/// Move the TCP relative to a reference cartesian position (PTPT interpolation)
FUNCTION_BLOCK MoveDirectOffsetFB EXTENDS RobotLibraryBaseFB
// ------------------------------------------------------------------------- 
//  SRCI Robot Library                                                
// ------------------------------------------------------------------------- 
//                                                                           
//  Object:      MoveDirectOffsetFB                                       
//  Author:      Thorsten Brach                                                
//  Date:        2024-06-01
//
//  Description:                                              
//   
//                                                                           
//  Copyright: 
//    (C) 2024 Thorsten Brach. All rights reserved                                                                         
//                                                                           
//  Disclaimer:                                                                           
//    This project is provided without any guarantee and can be used for   
//    private and commercial purposes. Any commercial use is at the user’s 
//    own risk and responsibility.
//
// -------------------------------------------------------------------------
VAR_INPUT
  /// Start of the command at the rising edge
  Execute            : BOOL;
  /// Absolute reference coordinates in the selected coordinate system (see input parameters ToolNo and FrameNo).
  ReferencePosition  : RobotCartesianPosition;
  /// Relative distance and rotation from ReferencePosition.
  Offset             : RobotCartesianPosition;
  /// Defines type of reference coordinate system of the offset position
  ReferenceType      : ReferenceType;
  /// TCP velocity in % of nominal velocity
  /// •  <0%: (default) - Use default velocity
  /// •   0%:           - Use internal minimal velocity
  /// • 100%:           - Use maximal reference velocity
  /// See chapter 5.5.7 Robot dynamics
  VelocityRate       : REAL;
  /// Acceleration for movement in % of nominal acceleration
  /// •  <0%: (default) - Use default acceleration
  /// •   0%:           - Use internal minimal acceleration
  /// • 100%:           - Use maximal reference acceleration
  /// See chapter 5.5.7 Robot dynamics
  AccelerationRate   : REAL;
  /// Deceleration for movement in % of nominal deceleration
  /// •  <0%: (default) - Use default deceleration 
  /// •   0%:           - Use internal minimal deceleration
  /// • 100%:           - Use maximal reference deceleration
  /// See chapter 5.5.7 Robot dynamics
  DecelerationRate   : REAL;
  /// Jerk of the movement in % of nominal jerk
  /// •  <0%: (default) - Use default jerk
  /// •   0%:           - Use internal minimal jerk
  /// • 100%:           - Use maximal reference jerk
  /// See chapter 5.5.7 Robot dynamics
  JerkRate           : REAL;
  /// Index of tool
  /// •      0: Flange (default)
  /// • 1..254: Tool frames
  ToolNo             : USINT;
  /// Index of frame
  /// •      0: WCS (default)
  /// • 1..254: User frames
  FrameNo            : USINT;
  /// Parameter which determines the behavior towards the previously sent and still active or buffered commands
  AbortingMode       : AbortingMode;
  /// Parameter which determines the transition behavior at the end of the movement to be sent to the next command. 
  /// The user can choose a transition type between exact stop and different blend possibilities
  BlendingMode       : BlendingMode;
  /// Additional parameter for the blending mode, to define i.e. velocity limit (%) or blending radius
  BlendingParameter  : ARRAY [0..1] OF REAL := [10,0];
  /// Parameter is used if it is greater than 0 (default)
  /// • Velocity input is ignored
  /// • Parameter defines the time for the movement to reach the target position
  /// Error is sent by the RC if the time cannot be kept
  MoveTime           : TIME;
  /// Parameter to describe how the orientation axes (RX, RY, RZ) will be interpolated during the movement.
  OriMode            : OriMode;
  /// Defines the usage of the config byte inside the position according to Table 6-238
  ConfigMode         : ArmConfigParameter;
  /// Defines the usage of the TurnNumber byte inside the position.
  TurnMode           : TurnMode;
  /// Set TRUE to allow manipulation of this move command through superimposing functions.
  /// For more information see chapter 5.5.9.5
  Manipulation       : BOOL;
  /// Defines the target sequence in which the command will be executed
  SequenceFlag       : SequenceFlag;
  /// ID of Action that will be executed when this command is active
  /// • >0: Start Action - Start executing the Action function with the identical ListenerID.
  /// • <0: Stop Action  -  Stop executing the Action function with the identical ListenerID.
  /// • 0: No trigger (default)-  If no EmitterID is defined, the function will not trigger any Action during its execution
  /// For more information see section Triggers of this chapter or chapter 5.5.12.4.
  EmitterID          : ARRAY [0..3] OF SINT;
END_VAR

VAR_OUTPUT
  /// The command has been completed successfully
  Done               : BOOL;
  /// FB is being processed
  Busy               : BOOL;
  /// Command is transferred and confirmed by the RC
  CommandBuffered    : BOOL;
  /// The command takes control of the motion of the according axis group
  Active             : BOOL;
  /// The command was aborted by another command.
  CommandAborted     : BOOL;
  /// TRUE, while command is interrupted during execution and can be continued
  CommandInterrupted : BOOL;
  /// Distance-to-go of the current job.
  /// • -1: No valid value because move command is not yet active (valid values are pending) or not supported by RC
  /// • >0: Actual distance between current and target position
  /// •  0: Target position reached
  RemainingDistance  : REAL;
  /// Percentage of already traversed distance of current job.
  /// If not supported : • -1
  Progress           : REAL;
  /// Unique system-generated ID of the trigger function when the function is called by the user.
  /// For more information see chapter 5.5.12.4.
  FollowID           : DINT;
END_VAR

                  
                

METHOD PROTECTED OnCall
VAR_IN_OUT
  /// Robot assignment of function
  AxesGroup         : AxesGroup; 
END_VAR
                        
                      
END_METHOD
END_FUNCTION_BLOCK

/// Move Joints relative to relative cartesian position (Relative cartesian PTP) (Joint interpolated movement)
FUNCTION_BLOCK MoveDirectRelativeFB EXTENDS RobotLibraryBaseFB
// ------------------------------------------------------------------------- 
//  SRCI Robot Library                                                
// ------------------------------------------------------------------------- 
//                                                                           
//  Object:      MoveDirectRelativeFB                                       
//  Author:      Thorsten Brach                                                
//  Date:        2024-06-01
//
//  Description:                                              
//   
//                                                                           
//  Copyright: 
//    (C) 2024 Thorsten Brach. All rights reserved                                                                         
//                                                                           
//  Disclaimer:                                                                           
//    This project is provided without any guarantee and can be used for   
//    private and commercial purposes. Any commercial use is at the user’s 
//    own risk and responsibility.
//
// -------------------------------------------------------------------------
VAR_INPUT
  /// Start of the command at the rising edge
  Execute            : BOOL;
  /// Relative distance and rotation from the current or last target position to the end point.
  Distance           : RobotCartesianPosition;
  /// Defines type of reference coordinate system of the offset position 
  ReferenceType      : ReferenceType;
  /// TCP velocity in % of nominal velocity
  /// •  <0%: (default) - Use default velocity
  /// •   0%:           - Use internal minimal velocity
  /// • 100%:           - Use maximal reference velocity
  /// See chapter 5.5.7 Robot dynamics
  ///
  VelocityRate       : REAL;
  /// Acceleration for movement in % of nominal acceleration
  /// •  <0%: (default) - Use default acceleration
  /// •   0%:           - Use internal minimal acceleration
  /// • 100%:           - Use maximal reference acceleration
  /// See chapter 5.5.7 Robot dynamics
  AccelerationRate   : REAL;
  /// Deceleration for movement in % of nominal deceleration
  /// •  <0%: (default) - Use default deceleration 
  /// •   0%:           - Use internal minimal deceleration
  /// • 100%:           - Use maximal reference deceleration
  /// See chapter 5.5.7 Robot dynamics
  DecelerationRate   : REAL;
  /// Jerk of the movement in % of nominal jerk
  /// •  <0%: (default) - Use default jerk
  /// •   0%:           - Use internal minimal jerk
  /// • 100%:           - Use maximal reference jerk
  /// See chapter 5.5.7 Robot dynamics
  JerkRate           : REAL;
  /// Index of tool
  /// •      0: Flange (default)
  /// • 1..254: Tool frames
  ToolNo             : USINT;
  /// Index of frame
  /// •      0: WCS (default)
  /// • 1..254: User frames
  FrameNo            : USINT;
  /// Parameter which determines the behavior towards the previously sent and still active or buffered commands
  AbortingMode       : AbortingMode;
  /// Parameter which determines the transition behavior at the end of the movement to be sent to the next command. 
  /// The user can choose a transition type between exact stop and different blend possibilities
  BlendingMode       : BlendingMode;
  /// Additional parameter for the blending mode, to define i.e. velocity limit (%) or blending radius
  BlendingParameter  : ARRAY [0..1] OF REAL := [10,0];
  /// Parameter is used if it is greater than 0 (default)
  /// • Velocity input is ignored
  /// • Parameter defines the time for the movement to reach the target position
  /// Error is sent by the RC if the time cannot be kept
  MoveTime           : TIME;
  /// Defines the usage of the config byte inside the position according to Table 6-238
  ConfigMode         : ArmConfigParameter;
  /// Defines the usage of the TurnNumber byte inside the position.
  TurnMode           : TurnMode;
  /// Set TRUE to allow manipulation of this move command through superimposing functions.
  /// For more information see chapter 5.5.9.5
  Manipulation       : BOOL;
  /// Defines the target sequence in which the command will be executed
  SequenceFlag       : SequenceFlag;
  /// ID of Action that will be executed when this command is active
  /// • >0: Start Action - Start executing the Action function with the identical ListenerID.
  /// • <0: Stop Action  -  Stop executing the Action function with the identical ListenerID.
  /// • 0: No trigger (default)-  If no EmitterID is defined, the function will not trigger any Action during its execution
  /// For more information see section Triggers of this chapter or chapter 5.5.12.4.
  EmitterID          : ARRAY [0..3] OF SINT;
END_VAR

VAR_OUTPUT
  /// The command has been completed successfully
  Done               : BOOL;
  /// FB is being processed
  Busy               : BOOL;
  /// Command is transferred and confirmed by the RC
  CommandBuffered    : BOOL;
  /// The command takes control of the motion of the according axis group
  Active             : BOOL;
  /// The command was aborted by another command.
  CommandAborted     : BOOL;
  /// TRUE, while command is interrupted during execution and can be continued
  CommandInterrupted : BOOL;
  /// Distance-to-go of the current job.
  /// • -1: No valid value because move command is not yet active (valid values are pending) or not supported by RC
  /// • >0: Actual distance between current and target position
  /// •  0: Target position reached
  RemainingDistance  : REAL;
  /// Percentage of already traversed distance of current job.
  /// If not supported : • -1
  Progress           : REAL;
  /// Unique system-generated ID of the trigger function when the function is called by the user.
  /// For more information see chapter 5.5.12.4.
  FollowID           : DINT;
END_VAR

                  
                

METHOD PROTECTED OnCall
VAR_IN_OUT
  /// Robot assignment of function
  AxesGroup         : AxesGroup; 
END_VAR
                        
                      
END_METHOD
END_FUNCTION_BLOCK

/// Move the TCP to an absolute cartesian position (linear interpolation)
FUNCTION_BLOCK MoveLinearAbsoluteFB EXTENDS RobotLibraryBaseFB
// ------------------------------------------------------------------------- 
//  SRCI Robot Library                                                
// ------------------------------------------------------------------------- 
//                                                                           
//  Object:      MoveLinearAbsoluteFB                                       
//  Author:      Thorsten Brach                                                
//  Date:        2024-06-01
//
//  Description:                                              
//   
//                                                                           
//  Copyright: 
//    (C) 2024 Thorsten Brach. All rights reserved                                                                         
//                                                                           
//  Disclaimer:                                                                           
//    This project is provided without any guarantee and can be used for   
//    private and commercial purposes. Any commercial use is at the user’s 
//    own risk and responsibility.
//
// -------------------------------------------------------------------------
VAR_INPUT
  /// Start of the command at the rising edge
  Execute            : BOOL;
  /// Absolute target coordinates in the selected coordinate system (see input parameters ToolNo and FrameNo)
  Position           : RobotCartesianPosition;
  /// TCP velocity in % of nominal velocity
  /// •  <0%: (default) - Use default velocity
  /// •   0%:           - Use internal minimal velocity
  /// • 100%:           - Use maximal reference velocity
  /// See chapter 5.5.7 Robot dynamics
  VelocityRate       : REAL;
  /// Acceleration for movement in % of nominal acceleration
  /// •  <0%: (default) - Use default acceleration
  /// •   0%:           - Use internal minimal acceleration
  /// • 100%:           - Use maximal reference acceleration
  /// See chapter 5.5.7 Robot dynamics
  AccelerationRate   : REAL;
  /// Deceleration for movement in % of nominal deceleration
  /// •  <0%: (default) - Use default deceleration 
  /// •   0%:           - Use internal minimal deceleration
  /// • 100%:           - Use maximal reference deceleration
  /// See chapter 5.5.7 Robot dynamics
  DecelerationRate   : REAL;
  /// Jerk of the movement in % of nominal jerk
  /// •  <0%: (default) - Use default jerk
  /// •   0%:           - Use internal minimal jerk
  /// • 100%:           - Use maximal reference jerk
  /// See chapter 5.5.7 Robot dynamics
  JerkRate           : REAL;
  /// Index of tool
  /// •      0: Flange (default)
  /// • 1..254: Tool frames
  ToolNo             : USINT;
  /// Index of frame
  /// •      0: WCS (default)
  /// • 1..254: User frames
  FrameNo            : USINT;
  /// Parameter which determines the behavior towards the previously sent and still active or buffered commands
  AbortingMode       : AbortingMode;
  /// Parameter which determines the transition behavior at the end of the movement to be sent to the next command. 
  /// The user can choose a transition type between exact stop and different blend possibilities
  BlendingMode       : BlendingMode;
  /// Additional parameter for the blending mode, to define i.e. velocity limit (%) or blending radius
  BlendingParameter  : ARRAY [0..1] OF REAL := [10,0];
  /// Parameter is used if it is greater than 0 (default)
  /// • Velocity input is ignored
  /// • Parameter defines the time for the movement to reach the target position
  /// Error is sent by the RC if the time cannot be kept
  MoveTime           : TIME;
  /// Parameter to describe how the orientation axes (RX, RY, RZ) will be interpolated during the movement
  OriMode            : OriMode;
  /// Defines the usage of the config byte inside the position according to Table 6-238
  ConfigMode         : ArmConfigParameter;
  /// Defines the usage of the TurnNumber byte inside the position.
  TurnMode           : TurnMode;
  /// Set TRUE to allow manipulation of this move command through superimposing functions.
  /// For more information see chapter 5.5.9.5
  Manipulation       : BOOL;
  /// Defines the target sequence in which the command will be executed
  SequenceFlag       : SequenceFlag;
  /// ID of Action that will be executed when this command is active
  /// • >0: Start Action - Start executing the Action function with the identical ListenerID.
  /// • <0: Stop Action  -  Stop executing the Action function with the identical ListenerID.
  /// • 0: No trigger (default)-  If no EmitterID is defined, the function will not trigger any Action during its execution
  /// For more information see section Triggers of this chapter or chapter 5.5.12.4.
  EmitterID          : ARRAY [0..3] OF SINT;
END_VAR

VAR_OUTPUT
  /// The command has been completed successfully
  Done               : BOOL;
  /// FB is being processed
  Busy               : BOOL;
  /// Command is transferred and confirmed by the RC
  CommandBuffered    : BOOL;
  /// The command takes control of the motion of the according axis group
  Active             : BOOL;
  /// The command was aborted by another command.
  CommandAborted     : BOOL;
  /// TRUE, while command is interrupted during execution and can be continued
  CommandInterrupted : BOOL;
  /// Distance-to-go of the current job.
  /// • -1: No valid value because move command is not yet active (valid values are pending) or not supported by RC
  /// • >0: Actual distance between current and target position
  /// •  0: Target position reached
  RemainingDistance  : REAL;
  /// Percentage of already traversed distance of current job.
  /// If not supported : • -1
  Progress           : REAL;
  /// Unique system-generated ID of the trigger function when the function is called by the user.
  /// For more information see chapter 5.5.12.4.
  FollowID           : DINT;
END_VAR

                  
                

METHOD PROTECTED OnCall
VAR_IN_OUT
  /// Robot assignment of function
  AxesGroup         : AxesGroup; 
END_VAR
                        
                      
END_METHOD
END_FUNCTION_BLOCK

/// Move TCP to an absolute joint position (linear interpolation)
FUNCTION_BLOCK MoveLinearAbsoluteJFB EXTENDS RobotLibraryBaseFB
// ------------------------------------------------------------------------- 
//  SRCI Robot Library                                                
// ------------------------------------------------------------------------- 
//                                                                           
//  Object:      MoveLinearAbsoluteJFB                                       
//  Author:      Thorsten Brach                                                
//  Date:        2024-06-01
//
//  Description:                                              
//   
//                                                                           
//  Copyright: 
//    (C) 2024 Thorsten Brach. All rights reserved                                                                         
//                                                                           
//  Disclaimer:                                                                           
//    This project is provided without any guarantee and can be used for   
//    private and commercial purposes. Any commercial use is at the user’s 
//    own risk and responsibility.
//
// -------------------------------------------------------------------------
VAR_INPUT
  /// Start of the command at the rising edge
  Execute            : BOOL;
  /// Absolute end position of the robot in Joint position.
  JointPosition      : RobotJointPosition;
  /// TCP velocity in % of nominal velocity
  /// •  <0%: (default) - Use default velocity
  /// •   0%:           - Use internal minimal velocity
  /// • 100%:           - Use maximal reference velocity
  /// See chapter 5.5.7 Robot dynamics
  VelocityRate       : REAL;
  /// Acceleration for movement in % of nominal acceleration
  /// •  <0%: (default) - Use default acceleration
  /// •   0%:           - Use internal minimal acceleration
  /// • 100%:           - Use maximal reference acceleration
  /// See chapter 5.5.7 Robot dynamics
  AccelerationRate   : REAL;
  /// Deceleration for movement in % of nominal deceleration
  /// •  <0%: (default) - Use default deceleration 
  /// •   0%:           - Use internal minimal deceleration
  /// • 100%:           - Use maximal reference deceleration
  /// See chapter 5.5.7 Robot dynamics
  DecelerationRate   : REAL;
  /// Jerk of the movement in % of nominal jerk
  /// •  <0%: (default) - Use default jerk
  /// •   0%:           - Use internal minimal jerk
  /// • 100%:           - Use maximal reference jerk
  /// See chapter 5.5.7 Robot dynamics
  JerkRate           : REAL;
  /// Index of tool
  /// •      0: Flange (default)
  /// • 1..254: Tool frames
  ToolNo             : USINT;
  /// Parameter which determines the behavior towards the previously sent and still active or buffered commands
  AbortingMode       : AbortingMode;
  /// Parameter which determines the transition behavior at the end of the movement to be sent to the next command. 
  /// The user can choose a transition type between exact stop and different blend possibilities
  BlendingMode       : BlendingMode;
  /// Additional parameter for the blending mode, to define i.e. velocity limit (%) or blending radius
  BlendingParameter  : ARRAY [0..1] OF REAL := [10,0];
  /// Parameter is used if it is greater than 0 (default)
  /// • Velocity input is ignored
  /// • Parameter defines the time for the movement to reach the target position
  /// Error is sent by the RC if the time cannot be kept
  MoveTime           : TIME;
  /// Parameter to describe how the orientation axes (RX, RY, RZ) will be interpolated during the movement
  OriMode            : OriMode;
  /// Set TRUE to allow manipulation of this move command through superimposing functions.
  /// For more information see chapter 5.5.9.5
  Manipulation       : BOOL;
  /// Defines the target sequence in which the command will be executed
  SequenceFlag       : SequenceFlag;
  /// ID of Action that will be executed when this command is active
  /// • >0: Start Action - Start executing the Action function with the identical ListenerID.
  /// • <0: Stop Action  -  Stop executing the Action function with the identical ListenerID.
  /// • 0: No trigger (default)-  If no EmitterID is defined, the function will not trigger any Action during its execution
  /// For more information see section Triggers of this chapter or chapter 5.5.12.4.
  EmitterID          : ARRAY [0..3] OF SINT;
END_VAR

VAR_OUTPUT
  /// The command has been completed successfully
  Done               : BOOL;
  /// FB is being processed
  Busy               : BOOL;
  /// Command is transferred and confirmed by the RC
  CommandBuffered    : BOOL;
  /// The command takes control of the motion of the according axis group
  Active             : BOOL;
  /// The command was aborted by another command.
  CommandAborted     : BOOL;
  /// TRUE, while command is interrupted during execution and can be continued
  CommandInterrupted : BOOL;
  /// Distance-to-go of the current job.
  /// • -1: No valid value because move command is not yet active (valid values are pending) or not supported by RC
  /// • >0: Actual distance between current and target position
  /// •  0: Target position reached
  RemainingDistance  : REAL;
  /// Percentage of already traversed distance of current job.
  /// If not supported : • -1
  Progress           : REAL;
  /// Unique system-generated ID of the trigger function when the function is called by the user.
  /// For more information see chapter 5.5.12.4.
  FollowID           : DINT;
END_VAR

                  
                

METHOD PROTECTED OnCall
VAR_IN_OUT
  /// Robot assignment of function
  AxesGroup         : AxesGroup; 
END_VAR
                        
                      
END_METHOD
END_FUNCTION_BLOCK

/// Set trigger in defined position of path (L = Linear Path) (cartesian) switch periphery.
FUNCTION_BLOCK MoveLinearCamFB EXTENDS RobotLibraryBaseFB
// ------------------------------------------------------------------------- 
//  SRCI Robot Library                                                
// ------------------------------------------------------------------------- 
//                                                                           
//  Object:      MoveLinearCamFB                                       
//  Author:      Thorsten Brach                                                
//  Date:        2024-06-01
//
//  Description:                                              
//   
//                                                                           
//  Copyright: 
//    (C) 2024 Thorsten Brach. All rights reserved                                                                         
//                                                                           
//  Disclaimer:                                                                           
//    This project is provided without any guarantee and can be used for   
//    private and commercial purposes. Any commercial use is at the user’s 
//    own risk and responsibility.
//
// -------------------------------------------------------------------------
VAR_INPUT
  /// Start of the command at the rising edge
  Execute            : BOOL;
  /// Absolute target coordinates in the selected coordinate system (see input parameters ToolNo and FrameNo)
  Position           : RobotCartesianPosition;
  /// TCP velocity in % of nominal velocity
  /// •  <0%: (default) - Use default velocity
  /// •   0%:           - Use internal minimal velocity
  /// • 100%:           - Use maximal reference velocity
  /// See chapter 5.5.7 Robot dynamics
  VelocityRate       : REAL;
  /// Acceleration for movement in % of nominal acceleration
  /// •  <0%: (default) - Use default acceleration
  /// •   0%:           - Use internal minimal acceleration
  /// • 100%:           - Use maximal reference acceleration
  /// See chapter 5.5.7 Robot dynamics
  AccelerationRate   : REAL;
  /// Deceleration for movement in % of nominal deceleration
  /// •  <0%: (default) - Use default deceleration 
  /// •   0%:           - Use internal minimal deceleration
  /// • 100%:           - Use maximal reference deceleration
  /// See chapter 5.5.7 Robot dynamics
  DecelerationRate   : REAL;
  /// Jerk of the movement in % of nominal jerk
  /// •  <0%: (default) - Use default jerk
  /// •   0%:           - Use internal minimal jerk
  /// • 100%:           - Use maximal reference jerk
  /// See chapter 5.5.7 Robot dynamics
  JerkRate           : REAL;
  /// Index of tool
  /// •      0: Flange (default)
  /// • 1..254: Tool frames
  ToolNo             : USINT;
  /// Index of frame
  /// •      0: WCS (default)
  /// • 1..254: User frames
  FrameNo            : USINT;
  /// Parameter which determines the behavior towards the previously sent and still active or buffered commands
  AbortingMode       : AbortingMode;
  /// Parameter which determines the transition behavior at the end of the movement to be sent to the next command. 
  /// The user can choose a transition type between exact stop and different blend possibilities
  BlendingMode       : BlendingMode;
  /// Additional parameter for the blending mode, to define i.e. velocity limit (%) or blending radius
  BlendingParameter  : ARRAY [0..1] OF REAL := [10,0];
  /// Parameter is used if it is greater than 0 (default)
  /// • Velocity input is ignored
  /// • Parameter defines the time for the movement to reach the target position
  /// Error is sent by the RC if the time cannot be kept
  MoveTime           : TIME;
  /// Parameter to describe how the orientation axes (RX, RY, RZ) will be interpolated during the movement
  OriMode            : OriMode;
  /// Defines the usage of the config byte inside the position according to Table 6-238
  ConfigMode         : ArmConfigParameter;
  /// Defines the usage of the TurnNumber byte inside the position.
  TurnMode           : TurnMode;
  /// Specifies the desired byte address that shall be written
  Index              : USINT;
  /// Specifies which output may be written
  OutputBitmask      : BYTE;
  /// Value of Digital Output
  Value              : BYTE;
  /// Reference position for the trigger point (at least one option must be supported):
  /// • 0: Start position (default) O
  /// • 1: End position
  RelativePosition   : BOOL;
  /// Time delay [ms] for the trigger point
  TriggerDelay       : UINT;
  /// Offset in millimeters towards the trigger point in relation to the reference position
  TriggerDistance    : REAL;
  /// Set TRUE to allow manipulation of this move command through superimposing functions.
  /// For more information see chapter 5.5.9.5
  Manipulation       : BOOL;
  /// Defines the target sequence in which the command will be executed
  SequenceFlag       : SequenceFlag;
END_VAR

VAR_OUTPUT
  /// The command has been completed successfully
  Done               : BOOL;
  /// FB is being processed
  Busy               : BOOL;
  /// Command is transferred and confirmed by the RC
  CommandBuffered    : BOOL;
  /// The command takes control of the motion of the according axis group
  Active             : BOOL;
  /// The command was aborted by another command.
  CommandAborted     : BOOL;
  /// TRUE, while command is interrupted during execution and can be continued
  CommandInterrupted : BOOL;
  /// Distance-to-go of the current job.
  /// • -1: No valid value because move command is not yet active (valid values are pending) or not supported by RC
  /// • >0: Actual distance between current and target position
  /// •  0: Target position reached
  RemainingDistance  : REAL;
  /// Percentage of already traversed distance of current job.
  /// If not supported : • -1
  Progress           : REAL;
END_VAR

                  
                

METHOD PROTECTED OnCall
VAR_IN_OUT
  /// Robot assignment of function
  AxesGroup         : AxesGroup; 
END_VAR
                        
                      
END_METHOD
END_FUNCTION_BLOCK

/// Move the TCP relative to a reference cartesian position (linear interpolation)
FUNCTION_BLOCK MoveLinearOffsetFB EXTENDS RobotLibraryBaseFB
// ------------------------------------------------------------------------- 
//  SRCI Robot Library                                                
// ------------------------------------------------------------------------- 
//                                                                           
//  Object:      MoveLinearOffsetFB                                       
//  Author:      Thorsten Brach                                                
//  Date:        2024-06-01
//
//  Description:                                              
//   
//                                                                           
//  Copyright: 
//    (C) 2024 Thorsten Brach. All rights reserved                                                                         
//                                                                           
//  Disclaimer:                                                                           
//    This project is provided without any guarantee and can be used for   
//    private and commercial purposes. Any commercial use is at the user’s 
//    own risk and responsibility.
//
// -------------------------------------------------------------------------
VAR_INPUT
  /// Start of the command at the rising edge
  Execute            : BOOL;
  /// Absolute reference coordinates in the selected coordinate system (see input parameters ToolNo and FrameNo).
  ReferencePosition  : RobotCartesianPosition;
  /// Relative distance and rotation from ReferencePosition.
  Offset             : RobotCartesianPosition;
  /// Defines type of reference coordinate system of the offset position.
  ReferenceType      : ReferenceType;
  /// TCP velocity in % of nominal velocity
  /// •  <0%: (default) - Use default velocity
  /// •   0%:           - Use internal minimal velocity
  /// • 100%:           - Use maximal reference velocity
  /// See chapter 5.5.7 Robot dynamics
  VelocityRate       : REAL;
  /// Acceleration for movement in % of nominal acceleration
  /// •  <0%: (default) - Use default acceleration
  /// •   0%:           - Use internal minimal acceleration
  /// • 100%:           - Use maximal reference acceleration
  /// See chapter 5.5.7 Robot dynamics
  AccelerationRate   : REAL;
  /// Deceleration for movement in % of nominal deceleration
  /// •  <0%: (default) - Use default deceleration 
  /// •   0%:           - Use internal minimal deceleration
  /// • 100%:           - Use maximal reference deceleration
  /// See chapter 5.5.7 Robot dynamics
  DecelerationRate   : REAL;
  /// Jerk of the movement in % of nominal jerk
  /// •  <0%: (default) - Use default jerk
  /// •   0%:           - Use internal minimal jerk
  /// • 100%:           - Use maximal reference jerk
  /// See chapter 5.5.7 Robot dynamics
  JerkRate           : REAL;
  /// Index of tool
  /// •      0: Flange (default)
  /// • 1..254: Tool frames
  ToolNo             : USINT;
  /// Index of frame
  /// •      0: WCS (default)
  /// • 1..254: User frames
  FrameNo            : USINT;
  /// Parameter which determines the behavior towards the previously sent and still active or buffered commands
  AbortingMode       : AbortingMode;
  /// Parameter which determines the transition behavior at the end of the movement to be sent to the next command. 
  /// The user can choose a transition type between exact stop and different blend possibilities
  BlendingMode       : BlendingMode;
  /// Additional parameter for the blending mode, to define i.e. velocity limit (%) or blending radius
  BlendingParameter  : ARRAY [0..1] OF REAL := [10,0];
  /// Parameter is used if it is greater than 0 (default)
  /// • Velocity input is ignored
  /// • Parameter defines the time for the movement to reach the target position
  /// Error is sent by the RC if the time cannot be kept
  MoveTime           : TIME;
  /// Parameter to describe how the orientation axes (RX, RY, RZ) will be interpolated during the movement
  OriMode            : OriMode;
  /// Defines the usage of the config byte inside the position according to Table 6-238
  ConfigMode         : ArmConfigParameter;
  /// Defines the usage of the TurnNumber byte inside the position.
  TurnMode           : TurnMode;
  /// Set TRUE to allow manipulation of this move command through superimposing functions.
  /// For more information see chapter 5.5.9.5
  Manipulation       : BOOL;
  /// Defines the target sequence in which the command will be executed
  SequenceFlag       : SequenceFlag;
  /// ID of Action that will be executed when this command is active
  /// • >0: Start Action - Start executing the Action function with the identical ListenerID.
  /// • <0: Stop Action  -  Stop executing the Action function with the identical ListenerID.
  /// • 0: No trigger (default)-  If no EmitterID is defined, the function will not trigger any Action during its execution
  /// For more information see section Triggers of this chapter or chapter 5.5.12.4.
  EmitterID          : ARRAY [0..3] OF SINT;
END_VAR

VAR_OUTPUT
  /// The command has been completed successfully
  Done               : BOOL;
  /// FB is being processed
  Busy               : BOOL;
  /// Command is transferred and confirmed by the RC
  CommandBuffered    : BOOL;
  /// The command takes control of the motion of the according axis group
  Active             : BOOL;
  /// The command was aborted by another command.
  CommandAborted     : BOOL;
  /// TRUE, while command is interrupted during execution and can be continued
  CommandInterrupted : BOOL;
  /// Distance-to-go of the current job.
  /// • -1: No valid value because move command is not yet active (valid values are pending) or not supported by RC
  /// • >0: Actual distance between current and target position
  /// •  0: Target position reached
  RemainingDistance  : REAL;
  /// Percentage of already traversed distance of current job.
  /// If not supported : • -1
  Progress           : REAL;
  /// Unique system-generated ID of the trigger function when the function is called by the user.
  /// For more information see chapter 5.5.12.4.
  FollowID           : DINT;
END_VAR

                  
                

METHOD PROTECTED OnCall
VAR_IN_OUT
  /// Robot assignment of function
  AxesGroup         : AxesGroup; 
END_VAR
                        
                      
END_METHOD
END_FUNCTION_BLOCK

/// Move the TCP relative to the actual cartesian position (linear interpolation)
FUNCTION_BLOCK MoveLinearRelativeFB EXTENDS RobotLibraryBaseFB
// ------------------------------------------------------------------------- 
//  SRCI Robot Library                                                
// ------------------------------------------------------------------------- 
//                                                                           
//  Object:      MoveLinearRelativeFB                                       
//  Author:      Thorsten Brach                                                
//  Date:        2024-06-01
//
//  Description:                                              
//   
//                                                                           
//  Copyright: 
//    (C) 2024 Thorsten Brach. All rights reserved                                                                         
//                                                                           
//  Disclaimer:                                                                           
//    This project is provided without any guarantee and can be used for   
//    private and commercial purposes. Any commercial use is at the user’s 
//    own risk and responsibility.
//
// -------------------------------------------------------------------------
VAR_INPUT
  /// Start of the command at the rising edge
  Execute            : BOOL;
  /// Relative distance and rotation from the current or last target position to the end point
  Distance           : RobotCartesianPosition;
  
  ReferenceType      : ReferenceType;
  /// TCP velocity in % of nominal velocity
  /// •  <0%: (default) - Use default velocity
  /// •   0%:           - Use internal minimal velocity
  /// • 100%:           - Use maximal reference velocity
  /// See chapter 5.5.7 Robot dynamics
  VelocityRate       : REAL;
  /// Acceleration for movement in % of nominal acceleration
  /// •  <0%: (default) - Use default acceleration
  /// •   0%:           - Use internal minimal acceleration
  /// • 100%:           - Use maximal reference acceleration
  /// See chapter 5.5.7 Robot dynamics
  AccelerationRate   : REAL;
  /// Deceleration for movement in % of nominal deceleration
  /// •  <0%: (default) - Use default deceleration 
  /// •   0%:           - Use internal minimal deceleration
  /// • 100%:           - Use maximal reference deceleration
  /// See chapter 5.5.7 Robot dynamics
  DecelerationRate   : REAL;
  /// Jerk of the movement in % of nominal jerk
  /// •  <0%: (default) - Use default jerk
  /// •   0%:           - Use internal minimal jerk
  /// • 100%:           - Use maximal reference jerk
  /// See chapter 5.5.7 Robot dynamics
  JerkRate           : REAL;
  /// Index of tool
  /// •      0: Flange (default)
  /// • 1..254: Tool frames
  ToolNo             : USINT;
  /// Index of frame
  /// •      0: WCS (default)
  /// • 1..254: User frames
  FrameNo            : USINT;
  /// Parameter which determines the behavior towards the previously sent and still active or buffered commands
  AbortingMode       : AbortingMode;
  /// Parameter which determines the transition behavior at the end of the movement to be sent to the next command. 
  /// The user can choose a transition type between exact stop and different blend possibilities
  BlendingMode       : BlendingMode;
  /// Additional parameter for the blending mode, to define i.e. velocity limit (%) or blending radius
  BlendingParameter  : ARRAY [0..1] OF REAL := [10,0];
  /// Parameter is used if it is greater than 0 (default)
  /// • Velocity input is ignored
  /// • Parameter defines the time for the movement to reach the target position
  /// Error is sent by the RC if the time cannot be kept
  MoveTime           : TIME;
  /// Parameter to describe how the orientation axes (RX, RY, RZ) will be interpolated during the movement
  OriMode            : OriMode;
  /// Defines the usage of the config byte inside the position according to Table 6-238
  ConfigMode         : ArmConfigParameter;
  /// Defines the usage of the TurnNumber byte inside the position.
  TurnMode           : TurnMode;
  /// Set TRUE to allow manipulation of this move command through superimposing functions.
  /// For more information see chapter 5.5.9.5
  Manipulation       : BOOL;
  /// Defines the target sequence in which the command will be executed
  SequenceFlag       : SequenceFlag;
  /// ID of Action that will be executed when this command is active
  /// • >0: Start Action - Start executing the Action function with the identical ListenerID.
  /// • <0: Stop Action  -  Stop executing the Action function with the identical ListenerID.
  /// • 0: No trigger (default)-  If no EmitterID is defined, the function will not trigger any Action during its execution
  /// For more information see section Triggers of this chapter or chapter 5.5.12.4.
  EmitterID          : ARRAY [0..3] OF SINT;
END_VAR

VAR_OUTPUT
  /// The command has been completed successfully
  Done               : BOOL;
  /// FB is being processed
  Busy               : BOOL;
  /// Command is transferred and confirmed by the RC
  CommandBuffered    : BOOL;
  /// The command takes control of the motion of the according axis group
  Active             : BOOL;
  /// The command was aborted by another command.
  CommandAborted     : BOOL;
  /// TRUE, while command is interrupted during execution and can be continued
  CommandInterrupted : BOOL;
  /// Distance-to-go [mm] of the current job
  /// • -1: No valid value because move command is not yet active (valid values are pending) or not supported by RC
  /// • >0: Actual distance between current and target position
  /// •  0: Target position reached
  RemainingDistance  : REAL;
  /// Percentage of already traversed distance of current job.
  /// If not supported : • -1
  Progress           : REAL;
  /// Unique system-generated ID of the trigger function when the function is called by the user.
  /// For more information see chapter 5.5.12.4.
  FollowID           : DINT;
END_VAR

                  
                

METHOD PROTECTED OnCall
VAR_IN_OUT
  /// Robot assignment of function
  AxesGroup         : AxesGroup; 
END_VAR
                        
                      
END_METHOD
END_FUNCTION_BLOCK

/// Commands interpolated movement of robot arm on a partly undefined path from actual position
FUNCTION_BLOCK MovePickPlaceDirectFB EXTENDS RobotLibraryBaseFB
// ------------------------------------------------------------------------- 
//  SRCI Robot Library                                                
// ------------------------------------------------------------------------- 
//                                                                           
//  Object:      MovePickPlaceDirectFB                                       
//  Author:      Thorsten Brach                                                
//  Date:        2024-06-01
//
//  Description:                                              
//   
//                                                                           
//  Copyright: 
//    (C) 2024 Thorsten Brach. All rights reserved                                                                         
//                                                                           
//  Disclaimer:                                                                           
//    This project is provided without any guarantee and can be used for   
//    private and commercial purposes. Any commercial use is at the user’s 
//    own risk and responsibility.
//
// -------------------------------------------------------------------------
VAR_INPUT
  /// Start of the command at the rising edge
  Execute            : BOOL;
  /// Absolute target coordinates in the selected coordinate system (see input parameters ToolNo and FrameNo)
  Position           : RobotCartesianPosition;
  /// Offset distance of auxiliary position from TargetPosition
  ApproachOffset     : AuxOffset;
  ///  Offset distance of auxiliary position from actual Position
  DepartOffset       : AuxOffset;
  /// Defines type of reference coordinate system of the offset position
  ReferenceType      : ReferenceType;
  /// TCP velocity in % of nominal velocity
  /// •  <0%: (default) - Use default velocity
  /// •   0%:           - Use internal minimal velocity
  /// • 100%:           - Use maximal reference velocity
  /// See chapter 5.5.7 Robot dynamics
  VelocityRate       : REAL;
  /// Acceleration for movement in % of nominal acceleration
  /// •  <0%: (default) - Use default acceleration
  /// •   0%:           - Use internal minimal acceleration
  /// • 100%:           - Use maximal reference acceleration
  /// See chapter 5.5.7 Robot dynamics
  AccelerationRate   : REAL;
  /// Deceleration for movement in % of nominal deceleration
  /// •  <0%: (default) - Use default deceleration 
  /// •   0%:           - Use internal minimal deceleration
  /// • 100%:           - Use maximal reference deceleration
  /// See chapter 5.5.7 Robot dynamics
  DecelerationRate   : REAL;
  /// Jerk of the movement in % of nominal jerk
  /// •  <0%: (default) - Use default jerk
  /// •   0%:           - Use internal minimal jerk
  /// • 100%:           - Use maximal reference jerk
  /// See chapter 5.5.7 Robot dynamics
  JerkRate           : REAL;
  /// Index of tool
  /// •      0: Flange (default)
  /// • 1..254: Tool frames
  ToolNo             : USINT;
  /// Index of frame
  /// •      0: WCS (default)
  /// • 1..254: User frames
  FrameNo            : USINT;
  /// Parameter which determines the behavior towards the previously sent and still active or buffered commands
  AbortingMode       : AbortingMode;
  /// Define blending sphere with radius around auxiliary position 1. For exact stop define AuxCornerDistance = 0
  AuxCornerDistance_1 : REAL;
  /// Define blending sphere with radius around auxiliary position 2. For exact stop define AuxCornerDistance = 0
  AuxCornerDistance_2 : REAL;
  /// Parameter is used if it is greater than 0 (default)
  /// • Velocity input is ignored
  /// • Parameter defines the time for the movement to reach the target position
  /// Error is sent by the RC if the time cannot be kept
  MoveTime           : TIME;
  /// Parameter to describe how the orientation axes (RX, RY, RZ) will be interpolated during the movement
  OriMode            : OriMode;
  /// Defines the usage of the config byte inside the position according to Table 6-238
  ConfigMode         : ArmConfigParameter;
  /// Defines the usage of the TurnNumber byte inside the position.
  TurnMode           : TurnMode;
  /// Factor by which VelocityRate is multiplied to define the velocity for the linear segments of the motion. Always positive.
  /// • 0: use the minimal velocity
  /// • 1: use the velocity set with VelocityRate
  /// Input values below 1 to reduce velocity.
  /// Input values above 1 to increase velocity.
  /// See chapter 5.5.7 Robot dynamics
  VelocityCoefficient: REAL;
  /// TCP velocity in % of the velocity set with VelocityRate to define the velocity for the linear motions. Always positive.
  /// • 0%: use the minimal velocity
  /// • 100%: use the velocity set with VelocityRate
  ReductionRate      : REAL;
  /// Set TRUE to allow manipulation of this move command through superimposing functions.
  /// For more information see chapter 5.5.9.5
  Manipulation       : BOOL;
  /// Defines the target sequence in which the command will be executed
  SequenceFlag       : SequenceFlag;
  /// ID of Action that will be executed when this command is active
  /// • >0: Start Action - Start executing the Action function with the identical ListenerID.
  /// • <0: Stop Action  -  Stop executing the Action function with the identical ListenerID.
  /// • 0: No trigger (default)-  If no EmitterID is defined, the function will not trigger any Action during its execution
  /// For more information see section Triggers of this chapter or chapter 5.5.12.4.
  EmitterID          : ARRAY [0..3] OF SINT;
END_VAR

VAR_OUTPUT
  /// The command has been completed successfully
  Done               : BOOL;
  /// FB is being processed
  Busy               : BOOL;
  /// Command is transferred and confirmed by the RC
  CommandBuffered    : BOOL;
  /// The command takes control of the motion of the according axis group
  Active             : BOOL;
  /// The command was aborted by another command.
  CommandAborted     : BOOL;
  /// TRUE, while command is interrupted during execution and can be continued
  CommandInterrupted : BOOL;
  /// Distance-to-go of the current job.
  /// • -1: No valid value because move command is not yet active (valid values are pending) or not supported by RC
  /// • >0: Actual distance between current and target position
  /// •  0: Target position reached
  RemainingDistance  : REAL;
  /// Percentage of already traversed distance of current job.
  /// If not supported : • -1
  Progress           : REAL;
  /// Unique system-generated ID of the trigger function when the function is called by the user.
  /// For more information see chapter 5.5.12.4.
  FollowID           : DINT;
END_VAR

                  
                

METHOD PROTECTED OnCall
VAR_IN_OUT
  /// Robot assignment of function
  AxesGroup         : AxesGroup; 
END_VAR
                        
                      
END_METHOD
END_FUNCTION_BLOCK

/// Command several interpolated movement of robot arm on linear paths from actual position
FUNCTION_BLOCK MovePickPlaceLinearFB EXTENDS RobotLibraryBaseFB
// ------------------------------------------------------------------------- 
//  SRCI Robot Library                                                
// ------------------------------------------------------------------------- 
//                                                                           
//  Object:      MovePickPlaceLinearFB                                       
//  Author:      Thorsten Brach                                                
//  Date:        2024-06-01
//
//  Description:                                              
//   
//                                                                           
//  Copyright: 
//    (C) 2024 Thorsten Brach. All rights reserved                                                                         
//                                                                           
//  Disclaimer:                                                                           
//    This project is provided without any guarantee and can be used for   
//    private and commercial purposes. Any commercial use is at the user’s 
//    own risk and responsibility.
//
// -------------------------------------------------------------------------
VAR_INPUT
  /// Start of the command at the rising edge
  Execute            : BOOL;
  /// Absolute target coordinates in the selected coordinate system (see input parameters ToolNo and FrameNo)
  Position           : RobotCartesianPosition;
  /// Offset distance of auxiliary position from TargetPosition
  ApproachOffset     : AuxOffset;
  ///  Offset distance of auxiliary position from actual Position
  DepartOffset       : AuxOffset;
  /// Defines type of reference coordinate system of the offset position
  ReferenceType      : ReferenceType;

  /// TCP velocity in % of nominal velocity
  /// •  <0%: (default) - Use default velocity
  /// •   0%:           - Use internal minimal velocity
  /// • 100%:           - Use maximal reference velocity
  /// See chapter 5.5.7 Robot dynamics
  VelocityRate       : REAL;
  /// Acceleration for movement in % of nominal acceleration
  /// •  <0%: (default) - Use default acceleration
  /// •   0%:           - Use internal minimal acceleration
  /// • 100%:           - Use maximal reference acceleration
  /// See chapter 5.5.7 Robot dynamics
  AccelerationRate   : REAL;
  /// Deceleration for movement in % of nominal deceleration
  /// •  <0%: (default) - Use default deceleration 
  /// •   0%:           - Use internal minimal deceleration
  /// • 100%:           - Use maximal reference deceleration
  /// See chapter 5.5.7 Robot dynamics
  DecelerationRate   : REAL;
  /// Jerk of the movement in % of nominal jerk
  /// •  <0%: (default) - Use default jerk
  /// •   0%:           - Use internal minimal jerk
  /// • 100%:           - Use maximal reference jerk
  /// See chapter 5.5.7 Robot dynamics
  JerkRate           : REAL;
  /// Index of tool
  /// •      0: Flange (default)
  /// • 1..254: Tool frames
  ToolNo             : USINT;
  /// Index of frame
  /// •      0: WCS (default)
  /// • 1..254: User frames
  FrameNo            : USINT;
  /// Parameter which determines the behavior towards the previously sent and still active or buffered commands
  AbortingMode       : AbortingMode;
  /// Define blending sphere with radius around auxiliary position 1. For exact stop define AuxCornerDistance = 0
  AuxCornerDistance_1 : REAL;
  /// Define blending sphere with radius around auxiliary position 2. For exact stop define AuxCornerDistance = 0
  AuxCornerDistance_2 : REAL;
  /// Parameter is used if it is greater than 0 (default)
  /// • Velocity input is ignored
  /// • Parameter defines the time for the movement to reach the target position
  /// Error is sent by the RC if the time cannot be kept
  MoveTime           : TIME;
  /// Parameter to describe how the orientation axes (RX, RY, RZ) will be interpolated during the movement
  OriMode            : OriMode;
  /// Defines the usage of the config byte inside the position according to Table 6-238
  ConfigMode         : ArmConfigParameter;
  /// Defines the usage of the TurnNumber byte inside the position.
  TurnMode           : TurnMode;
  /// Set TRUE to allow manipulation of this move command through superimposing functions.
  /// For more information see chapter 5.5.9.5
  Manipulation       : BOOL;
  /// Defines the target sequence in which the command will be executed
  SequenceFlag       : SequenceFlag;
  /// ID of Action that will be executed when this command is active
  /// • >0: Start Action - Start executing the Action function with the identical ListenerID.
  /// • <0: Stop Action  -  Stop executing the Action function with the identical ListenerID.
  /// • 0: No trigger (default)-  If no EmitterID is defined, the function will not trigger any Action during its execution
  /// For more information see section Triggers of this chapter or chapter 5.5.12.4.
  EmitterID          : ARRAY [0..3] OF SINT;
END_VAR

VAR_OUTPUT
  /// The command has been completed successfully
  Done               : BOOL;
  /// FB is being processed
  Busy               : BOOL;
  /// Command is transferred and confirmed by the RC
  CommandBuffered    : BOOL;
  /// The command takes control of the motion of the according axis group
  Active             : BOOL;
  /// The command was aborted by another command.
  CommandAborted     : BOOL;
  /// TRUE, while command is interrupted during execution and can be continued
  CommandInterrupted : BOOL;
  /// Distance-to-go of the current job.
  /// • -1: No valid value because move command is not yet active (valid values are pending) or not supported by RC
  /// • >0: Actual distance between current and target position
  /// •  0: Target position reached
  RemainingDistance  : REAL;
  /// Percentage of already traversed distance of current job.
  /// If not supported : • -1
  Progress           : REAL;
  /// Unique system-generated ID of the trigger function when the function is called by the user.
  /// For more information see chapter 5.5.12.4.
  FollowID           : DINT;
END_VAR

                  
                

METHOD PROTECTED OnCall
VAR_IN_OUT
  /// Robot assignment of function
  AxesGroup         : AxesGroup; 
END_VAR
                        
                      
END_METHOD
END_FUNCTION_BLOCK

/// Move spline previously created on RC
FUNCTION_BLOCK MoveSplineFB EXTENDS RobotLibraryBaseFB
// ------------------------------------------------------------------------- 
//  SRCI Robot Library                                                
// ------------------------------------------------------------------------- 
//                                                                           
//  Object:      MoveSplineFB                                       
//  Author:      Thorsten Brach                                                
//  Date:        2024-06-01
//
//  Description:                                              
//   
//                                                                           
//  Copyright: 
//    (C) 2024 Thorsten Brach. All rights reserved                                                                         
//                                                                           
//  Disclaimer:                                                                           
//    This project is provided without any guarantee and can be used for   
//    private and commercial purposes. Any commercial use is at the user’s 
//    own risk and responsibility.
//
// -------------------------------------------------------------------------
VAR_INPUT
  /// Start of the command at the rising edge
  Execute            : BOOL;
  /// Index of the spline data set, on which the spline trajectory is based
  SplineID           : SINT;
  ///Parameter which determines the behavior towards the previously sent and still active or buffered commands
  AbortingMode       : AbortingMode;
  /// Parameter which determines the transition behavior at the end of the movement to be sent to the next command. 
  /// The user can choose a transition type between exact stop and different blend possibilities.
  BlendingMode       : BlendingMode;
  /// Additional parameter for the blending mode, to define i.e. velocity limit (%) or blending radius
  /// • [0]: default 10
  /// • [1]: default 0
  BlendingParameter  : ARRAY [0..1] OF REAL;
  /// Parameter is used if it is greater than 0 (default):
  /// • Velocity input is ignored
  /// • Parameter defines the time for the movement to reach the target position 
  /// Error is sent by the RC, if the time cannot be kept.
  MoveTime           : UINT;
  /// Defines the target sequence in which the command will be executed
  SequenceFlag       : SequenceFlag;
END_VAR
VAR_OUTPUT
  /// The command has been completed successfully
  Done               : BOOL;
  /// FB is being processed
  Busy               : BOOL;
  /// Command is transferred and confirmed by the RC
  CommandBuffered    : BOOL;
  /// The command takes control of the motion of the according axis group.
  Active             : BOOL;
  /// The command was aborted by another command
  CommandAborted     : BOOL;
  /// TRUE, while command is interrupted during execution and can be continued
  CommandInterrupted : BOOL;
  /// Distance-to-go of the current job.
  /// • -1: No valid value because move command is not yet active (valid values are pending) or not supported by RC
  /// • >0: Actual distance between current and target position
  /// •  0: Target position reached 
  RemainingDistance  : REAL;
  /// Percentage of already traversed distance of current job. 
  /// If not supported: -1
  Progress           : REAL;
  /// Index of the currently active segment of spline data set.
  ActualIndex        : SINT;
END_VAR

                  
                

METHOD PROTECTED OnCall
VAR_IN_OUT
  /// Robot assignment of function
  AxesGroup         : AxesGroup; 
END_VAR
                        
                      
END_METHOD
END_FUNCTION_BLOCK

/// Activate superimposed motion of TCP to defined motion
FUNCTION_BLOCK MoveSuperImposedFB EXTENDS RobotLibraryBaseFB
// ------------------------------------------------------------------------- 
//  SRCI Robot Library                                                
// ------------------------------------------------------------------------- 
//                                                                           
//  Object:      MoveSuperImposedFB                                       
//  Author:      Thorsten Brach                                                
//  Date:        2024-06-01
//
//  Description:                                              
//   
//                                                                           
//  Copyright: 
//    (C) 2024 Thorsten Brach. All rights reserved                                                                         
//                                                                           
//  Disclaimer:                                                                           
//    This project is provided without any guarantee and can be used for   
//    private and commercial purposes. Any commercial use is at the user’s 
//    own risk and responsibility.
//
// -------------------------------------------------------------------------
VAR_INPUT
  /// Start of the command at the rising edge
  Execute            : BOOL;
  /// Processing mode
  ProcessingMode     : ProcessingMode;
  /// Additional distance and orientation for superimposed positioning:
  Offset             : RobotCartesianPosition;
  /// Defines type of reference coordinate system of the offset position.
  ReferenceType      : ReferenceType;
  /// Value of the maximum velocity difference of the additional motion (not necessary reached).
  /// • > 0% Use specified value.
  /// • ≤ 0% Use the velocity defined by the move command that is superimposed. If no motion is active, use internal minimal velocity. (default)
 /// See chapter 5.5.7 Robot dynamics
  VelocityDiffRate   : REAL;
  /// Value of the maximum acceleration difference of the additional motion (not necessary reached).
  ///  •  <0% Use default acceleration (default)
  ///  •   0% Use internal minimal acceleration
  ///  • 100% Use maximal reference acceleration
  /// See chapter 5.5.7 Robot dynamics
  AccelerationDiffRate: REAL;
  /// Value of the maximum deceleration difference of the additional motion (not necessary reached).
  /// •  <0% Use default deceleration (default)
  /// •   0% Use internal minimal deceleration
  /// • 100% Use maximal reference deceleration
  /// See chapter 5.5.7 Robot dynamics
  DecelerationDiffRate: REAL;
  /// Value of the maximum jerk difference of the additional motion (not necessary reached).
  /// •  <0% Use default jerk (default) 
  /// •   0% Use internal minimal jerk
  /// • 100% Use maximal reference jerk
  /// See chapter 5.5.7 Robot dynamics
  JerkDiffRate        : REAL;
  /// Index of tool
  /// •      0: Flange (default)
  /// • 1..254: Tool frames
  ToolNo             : USINT;
  /// Index of frame
  /// •      0: WCS (default)
  /// • 1..254: User frames
  FrameNo            : USINT;
  /// ID of the trigger function that may be triggered:
  /// •  0: Immediately (default) - Start executing this function immediately.
  /// • >0: Trigger               - Start executing when the trigger function with the identical positive EmitterID is called
  ///                             - Stop executing when the trigger function with the identical negative EmitterID is called.
  /// For more information see chapter 5.5.12.4.
  ListenerID         : SINT;
END_VAR

VAR_OUTPUT
  /// The command has been completed successfully
  Done               : BOOL;
  /// FB is being processed
  Busy               : BOOL;
  /// Command is transferred and confirmed by the RC
  CommandBuffered    : BOOL;
  /// The command takes control of the motion of the according axis group
  Active             : BOOL;
  /// Receiving of input parameter values has been acknowledged by RC
  ParameterAccepted  : BOOL;
  /// Distance-to-go [mm] of the current job
  /// • -1: No valid value because move command is not yet active (valid values are pending) or not supported by RC
  /// • >0: Actual distance between current and target position
  /// •  0: Target position reached
  RemainingDistance  : REAL;
  /// Percentage of already traversed superimposed offset.
  /// If not supported : • -1
  Progress           : REAL;
  /// Unique system-generated ID of the "Action" when the function is executed.
  /// • >0: The "Action" is started by the identical FollowID.
  /// • <0: The "Action" is stopped by the identical FollowID.
  /// For more information see chapter 5.5.12.4 EmitterID, ListenerID, FollowID and OriginID
  OriginID           : INT;
  /// Relates to ListenerID >0
  /// Number of successful trigger -based command invocations
  /// For more information refer to chapter 5.5.12.4
  InvocationCounter  : USINT;
END_VAR

                  
                

METHOD PROTECTED OnCall
VAR_IN_OUT
  /// Robot assignment of function
  AxesGroup         : AxesGroup; 
END_VAR
                        
                      
END_METHOD
END_FUNCTION_BLOCK

/// Activate superimposed motion of TCP to defined motion
FUNCTION_BLOCK MoveSuperImposedDynamicFB EXTENDS RobotLibraryBaseFB
// ------------------------------------------------------------------------- 
//  SRCI Robot Library                                                
// ------------------------------------------------------------------------- 
//                                                                           
//  Object:      MoveSuperImposedDynamicFB                                       
//  Author:      Thorsten Brach                                                
//  Date:        2024-06-01
//
//  Description:                                              
//   
//                                                                           
//  Copyright: 
//    (C) 2024 Thorsten Brach. All rights reserved                                                                         
//                                                                           
//  Disclaimer:                                                                           
//    This project is provided without any guarantee and can be used for   
//    private and commercial purposes. Any commercial use is at the user’s 
//    own risk and responsibility.
//
// -------------------------------------------------------------------------
VAR_INPUT
  /// Start of the command at the rising edge
  Execute            : BOOL;
  /// Additional distance and orientation for superimposed positioning
  Offset             : RobotCartesianPosition;
  /// Defines type of reference coordinate system of the offset position.
  ReferenceType      : ReferenceType;
  /// Value of the maximum velocity difference of the additional motion (not necessary reached).
  /// • > 0% Use specified value.
  /// • ≤ 0% Use the velocity defined by the move command that is superimposed. If no motion is active, use internal minimal velocity. (default)
 /// See chapter 5.5.7 Robot dynamics
  VelocityDiffRate   : REAL;
  /// Value of the maximum acceleration difference of the additional motion (not necessary reached).
  ///  •  <0% Use default acceleration (default)
  ///  •   0% Use internal minimal acceleration
  ///  • 100% Use maximal reference acceleration
  /// See chapter 5.5.7 Robot dynamics
  AccelerationDiffRate: REAL;
  /// Value of the maximum deceleration difference of the additional motion (not necessary reached).
  /// •  <0% Use default deceleration (default)
  /// •   0% Use internal minimal deceleration
  /// • 100% Use maximal reference deceleration
  /// See chapter 5.5.7 Robot dynamics
  DecelerationDiffRate: REAL;
  /// Value of the maximum jerk difference of the additional motion (not necessary reached).
  /// •  <0% Use default jerk (default) 
  /// •   0% Use internal minimal jerk
  /// • 100% Use maximal reference jerk
  /// See chapter 5.5.7 Robot dynamics
  JerkDiffRate        : REAL;
  /// Index of tool
  /// •      0: Flange (default)
  /// • 1..254: Tool frames
  ToolNo             : USINT;
  /// Index of frame
  /// •      0: WCS (default)
  /// • 1..254: User frames
  FrameNo            : USINT;
  /// Define the interpolation mode for the superimposed motion
  InterpolationMode  : InterpolationMode;
END_VAR

VAR_OUTPUT
  /// FB is being processed
  Busy               : BOOL;
  /// Command is transferred and confirmed by the RC
  CommandBuffered    : BOOL;
  /// The command takes control of the motion of the according axis group
  Active             : BOOL;
  /// Receiving of input parameter values has been acknowledged by RC
  ParameterAccepted  : BOOL;
  /// Distance-to-go [mm] of the current job
  /// • -1: No valid value because move command is not yet active (valid values are pending) or not supported by RC
  /// • >0: Actual distance between current and target position
  /// •  0: Target position reached
  RemainingDistance  : REAL;
  /// Percentage of already traversed superimposed offset.
  /// If not supported : • -1
  Progress           : REAL;
  /// TRUE if the offset for superimposed positioning is reached.
  OffsetReached      : BOOL;
END_VAR

                  
                

METHOD PROTECTED OnCall
VAR_IN_OUT
  /// Robot assignment of function
  AxesGroup         : AxesGroup; 
END_VAR
                        
                      
END_METHOD
END_FUNCTION_BLOCK

/// Read the actual position – TCP: X…RZ + config/Turn, … Joint: (J1…E6)
FUNCTION_BLOCK ReadActualPositionFB EXTENDS RobotLibraryBaseFB
// ------------------------------------------------------------------------- 
//  SRCI Robot Library                                                
// ------------------------------------------------------------------------- 
//                                                                           
//  Object:      ReadActualPositionFB                                       
//  Author:      Thorsten Brach                                                
//  Date:        2024-06-01
//
//  Description:                                              
//   
//                                                                           
//  Copyright: 
//    (C) 2024 Thorsten Brach. All rights reserved                                                                         
//                                                                           
//  Disclaimer:                                                                           
//    This project is provided without any guarantee and can be used for   
//    private and commercial purposes. Any commercial use is at the user’s 
//    own risk and responsibility.
//
// -------------------------------------------------------------------------
VAR_INPUT
  /// Start of the command at the rising edge
  Execute            : BOOL;
  /// Processing mode - For more information see chapter 5.6.4.5.
  ProcessingMode     : ProcessingMode;
  /// Index of tool of returned position
  /// •     -1: Currently used tool on RC
  /// •      0: Flange (default)
  /// • 1..254: Tool frames
  ToolNo             : INT;
  /// Index of frame of returned position
  /// •     -1: Currently used frame on RC
  /// •      0: WCS (default)
  /// • 1..254: User frames
  FrameNo            : INT;
  /// Defines the target sequence in which the command will be executed
  SequenceFlag       : SequenceFlag;
  /// ID of associated trigger function
  /// •  0: No Trigger (default) -> No trigger related behavior
  /// • >0: Trigger              -> Start executing when the trigger function with the identical EmitterID is triggered.
  /// Always positive. For more information, see chapter 5.5.12 Triggers
  ListenerID         : SINT;
END_VAR

VAR_OUTPUT
  /// The command has been completed successfully
  Done               : BOOL;
  /// TRUE, while the following outputs return valid values
  /// • ActualCartesianPosition
  /// • ToolNoReturn
  /// • FrameNoReturn
  /// • ActualJointPosition
  Valid              : BOOL;
  /// FB is being processed
  Busy               : BOOL;
  /// Command is transferred and confirmed by the RC
  CommandBuffered    : BOOL;  
  /// The command was aborted by another command.
  CommandAborted     : BOOL;
  /// TRUE, while command is interrupted during execution and can be continued.
  CommandInterrupted : BOOL;
  /// Receiving of input parameter values has been acknowledged by RC
  ParameterAccepted  : BOOL;
  /// Relates to ListenerID >0 Number of successful trigger -based command invocations. For more information refer to chapter 5.5.12.4.
  InvocationCounter  : USINT;
  /// Unique system-generated ID of the "Action" when the function is triggered 
  /// • >0: The "Action" is started by the trigger function with identical FollowID.
  /// • <0: The "Action" is stopped BY the trigger function with identical FollowID.
  /// For more information see chapter 5.5.12.4
  OriginID           : INT;
END_VAR

                  
                

METHOD PROTECTED OnCall
VAR_IN_OUT
  /// Robot assignment of function
  AxesGroup         : AxesGroup; 
END_VAR
                        
                      
END_METHOD
END_FUNCTION_BLOCK

/// Read the actual position cyclically
FUNCTION_BLOCK ReadActualPositionCyclicFB EXTENDS RobotLibraryBaseFB
// ------------------------------------------------------------------------- 
//  SRCI Robot Library                                                
// ------------------------------------------------------------------------- 
//                                                                           
//  Object:      ReadActualPositionCyclicFB                                       
//  Author:      Thorsten Brach                                                
//  Date:        2024-06-01
//
//  Description:                                              
//   
//                                                                           
//  Copyright: 
//    (C) 2024 Thorsten Brach. All rights reserved                                                                         
//                                                                           
//  Disclaimer:                                                                           
//    This project is provided without any guarantee and can be used for   
//    private and commercial purposes. Any commercial use is at the user’s 
//    own risk and responsibility.
//
// -------------------------------------------------------------------------
VAR_INPUT
  /// Set TRUE (default) to cyclically transmit position data
  Enable                      : BOOL;
  /// Set TRUE (default) to activate cyclic transmission of cartesian position without external axes
  ReadCartesianPosition       : BOOL;
  /// Set TRUE to activate cyclic transmission of external axes values of cartesian position -  Default: False
  ReadExtCartesianPosition    : BOOL;
  ///Index of tool of returned position
  /// •     -1: Currently used tool on RC
  /// •      0: Flange (default)
  /// • 1..254: Tool frames
  ToolNo                      : INT;
  /// Index of frame of returned position
  /// •     -1: Currently used frame on RC
  /// •      0: WCS (default)
  /// • 1..254: User frames
  FrameNo                     : INT;
  /// Set TRUE (default) to activate cyclic transmission of joint position without external axes
  ReadJointPosition           : BOOL;
  /// Set TRUE to activate cyclic transmission of external axes values of joint position - Default: False
  ReadExtJointPosition        : BOOL;
END_VAR

VAR_OUTPUT
  /// FB is enabled
  Enabled                     : BOOL;
  /// FB is being processed
  Busy                        : BOOL;
  /// TRUE, while the output CartesianPosition returns valid values
  ReadingCartesianPosition    : BOOL;
  /// TRUE, while the output ExtCartesianPosition returns valid values
  ReadingExtCartesianPosition : BOOL;
  /// TRUE, while the output JointPosition returns valid values
  ReadingJointPosition        : BOOL;
  /// TRUE, while the output ExtJointPosition returns valid values
  ReadingExtJointPosition     : BOOL;
  /// Tool and frame index of currently used tool and frame according to Table 6-40
  CurrentCoordinateSystem     : CoordinateSystem;
  /// Cyclically returned, absolute coordinates of current position in selected coordinate systems (see input parameters ToolNo and FrameNo) 
  CartesianPosition           : RobotCartesianPositionShort;
  /// Cyclically returned, absolute cartesian position of the external axes of the robot
  CartesianPositionExt        : RobotCartesianPositionExt;
  /// Tool and frame index of returned position according to Table 6-40
  CoordinateSystem            : CoordinateSystem;
  /// Cyclically returned, absolute position of the robot in Joint position
  JointPosition               : RobotJointPositionShort;
  /// Cyclically returned, absolute joint position of the external axes of the robot
  JointPositionExt            : RobotJointPositionExt;
END_VAR

                  
                

METHOD PROTECTED OnCall
VAR_IN_OUT
  /// Robot assignment of function
  AxesGroup         : AxesGroup; 
END_VAR
                        
                      
END_METHOD
END_FUNCTION_BLOCK

/// Read actual TCP velocity
FUNCTION_BLOCK ReadActualTCPVelocityFB EXTENDS RobotLibraryBaseFB
// ------------------------------------------------------------------------- 
//  SRCI Robot Library                                                
// ------------------------------------------------------------------------- 
//                                                                           
//  Object:      ReadActualTCPVelocityFB                                       
//  Author:      Thorsten Brach                                                
//  Date:        2024-06-01
//
//  Description:                                              
//   
//                                                                           
//  Copyright: 
//    (C) 2024 Thorsten Brach. All rights reserved                                                                         
//                                                                           
//  Disclaimer:                                                                           
//    This project is provided without any guarantee and can be used for   
//    private and commercial purposes. Any commercial use is at the user’s 
//    own risk and responsibility.
//
// -------------------------------------------------------------------------
VAR_INPUT
    /// Start of the command at the rising edge
  Execute            : BOOL;
  /// Processing mode
  ProcessingMode     : ProcessingMode;
  /// Index of tool of returned velocity
  /// •      0: Flange (default)
  /// • 1..254: Tool frames
  ToolNo             : USINT;
  /// Index of frame
  /// •      0: WCS (default)
  /// • 1..254: User frames
  FrameNo            : USINT;
  /// Defines the target sequence in which the command will be executed 
  ///  For more information about the differentiation of sequences see chapter 5.5.3.4
  SequenceFlag       : SequenceFlag;
  /// ID of associated trigger function
  /// • 0: No Trigger (default) -> No trigger related behavior
  /// • >0: Trigger             -> Start executing when the trigger function with the identical EmitterID is triggered. 
  /// Always positive.
  /// For more information, see chapter 5.5.12 Triggers
  ListenerID         : SINT;
END_VAR

VAR_OUTPUT
  /// The command has been completed successfully
  Done               : BOOL;
  /// TRUE, while the following outputs return valid values:
  /// • ActualTCPVelocity
  /// • ToolNoReturn
  /// • FrameNoReturn
  Valid              : BOOL;
  /// FB is being processed
  Busy               : BOOL;
  /// The command was aborted by another command.
  CommandAborted     : BOOL;
  /// Command is transferred and confirmed by the RC
  CommandBuffered    : BOOL;
  /// TRUE, while command is interrupted during execution and can be continued
  CommandInterrupted : BOOL;
  /// Receiving of input parameter values has been acknowledged by RC
  ParameterAccepted  : BOOL;
  /// Absolute actual velocity of the robot’s TCP. [mm/s]
  ActualTCPVelocity  : REAL;
  /// Index of tool of returned velocity
  /// •      0: Flange
  /// • 1..254: Tool frames
  ToolNoReturn       : USINT;
  /// Index of frame of returned position
  /// •      0: WCS
  /// • 1..254: User frames
  FrameNoReturn      : USINT;
  /// Unique system-generated ID of the "Action" when the function is triggered
  /// • >0: The "Action" is started by the trigger function with identical FollowID.
  /// • <0: The "Action" is stopped by the trigger function with identical FollowID.
  /// For more information see chapter 5.5.12.4
  OriginID           : INT;
  /// Relates to ListenerID >0 Number of successful trigger -based command invocations 
  /// For more information refer to chapter 5.5.12.4
  InvocationCounter  : USINT;
END_VAR

                  
                

METHOD PROTECTED OnCall
VAR_IN_OUT
  /// Robot assignment of function
  AxesGroup         : AxesGroup; 
END_VAR
                        
                      
END_METHOD
END_FUNCTION_BLOCK

/// Read analog input of RC
FUNCTION_BLOCK ReadAnalogInputFB EXTENDS RobotLibraryBaseFB
// ------------------------------------------------------------------------- 
//  SRCI Robot Library                                                
// ------------------------------------------------------------------------- 
//                                                                           
//  Object:      ReadAnalogInputFB                                       
//  Author:      Thorsten Brach                                                
//  Date:        2024-06-01
//
//  Description:                                              
//   
//                                                                           
//  Copyright: 
//    (C) 2024 Thorsten Brach. All rights reserved                                                                         
//                                                                           
//  Disclaimer:                                                                           
//    This project is provided without any guarantee and can be used for   
//    private and commercial purposes. Any commercial use is at the user’s 
//    own risk and responsibility.
//
// -------------------------------------------------------------------------
VAR_INPUT
  /// Start of the command at the rising edge
  Execute            : BOOL;
  /// Processing Mode
  ProcessingMode     : ProcessingMode;
  /// Number of the analog input 1..32
  Index              : USINT; 
  /// Defines the target sequence in which the command will be executed
  SequenceFlag       : SequenceFlag;
  /// ID of associated trigger function:
  /// •  0: No Trigger (default)  No trigger related behavior
  /// • >0: Trigger - Start executing when the trigger function with the identical EmitterID is triggered.
  /// Always positive.
  /// For more information, see chapter 5.5.12 Triggers
  ListenerID         : SINT;
END_VAR
VAR_OUTPUT
  /// The command has been completed successfully
  Done               : BOOL;
  /// TRUE, while the following outputs return valid values:
  /// • Values
  Valid              : BOOL; 
  /// FB is being processed
  Busy               : BOOL;
  /// Command is transferred and confirmed by the RC
  CommandBuffered    : BOOL;
  /// The command was aborted by another command.
  CommandAborted     : BOOL;
  /// TRUE, while command is interrupted during execution and can be continued
  CommandInterrupted : BOOL;
  /// Receiving of input parameter values has been acknowledged by RC
  ParameterAccepted  : BOOL;
  /// Returned values of digital inputs
  /// Unit of returned Value
  Unit               : UnitType;
  Value              : REAL;
  /// Unique system-generated ID of the "Action" when the function is triggered.
  /// • >0: The "Action" is started by the trigger function with identical FollowID.
  /// • <0: The "Action" is stopped by the trigger function with identical FollowID.
  /// For more information see chapter 5.5.12.4.
  OriginID           : USINT;
  /// Relates to ListenerID >0 
  /// Number of successful trigger -based command invocations
  /// For more information refer to chapter 5.5.12.4.
  InvocationCounter  : USINT;
END_VAR

                  
                

METHOD PROTECTED OnCall
VAR_IN_OUT
  /// Robot assignment of function
  AxesGroup         : AxesGroup; 
END_VAR
                        
                      
END_METHOD
END_FUNCTION_BLOCK

/// Read DH (Denavit–Hartenberg) parameters of robot
FUNCTION_BLOCK ReadDHParameterFB EXTENDS RobotLibraryBaseFB
// ------------------------------------------------------------------------- 
//  SRCI Robot Library                                                
// ------------------------------------------------------------------------- 
//                                                                           
//  Object:      ReadDHParameterFB                                       
//  Author:      Thorsten Brach                                                
//  Date:        2024-06-01
//
//  Description:                                              
//   
//                                                                           
//  Copyright: 
//    (C) 2024 Thorsten Brach. All rights reserved                                                                         
//                                                                           
//  Disclaimer:                                                                           
//    This project is provided without any guarantee and can be used for   
//    private and commercial purposes. Any commercial use is at the user’s 
//    own risk and responsibility.
//
// -------------------------------------------------------------------------
VAR_INPUT
  /// Start of the command at the rising edge
  Execute            : BOOL;
  /// Determines if returned DH parameters use modified convention or classic convention.
  /// • 0: Classic convention (default)
  /// • 1: Modified convention
  ModifiedConvention : BOOL;  
END_VAR

VAR_OUTPUT
  /// The command has been completed successfully
  Done               : BOOL;
  /// FB is being processed
  Busy               : BOOL;
  /// Command is transferred and confirmed by the RC
  CommandBuffered    : BOOL;
  /// Denavit–Hartenberg parameter
  DHParameter        : DHParameter;
END_VAR

                  
                

METHOD PROTECTED OnCall
VAR_IN_OUT
  /// Robot assignment of function
  AxesGroup         : AxesGroup; 
END_VAR
                        
                      
END_METHOD
END_FUNCTION_BLOCK

/// Read digital input and output group of RC
FUNCTION_BLOCK ReadDigitalInputsFB EXTENDS RobotLibraryBaseFB
// ------------------------------------------------------------------------- 
//  SRCI Robot Library                                                
// ------------------------------------------------------------------------- 
//                                                                           
//  Object:      ReadDigitalInputsFB                                       
//  Author:      Thorsten Brach                                                
//  Date:        2024-06-01
//
//  Description:                                              
//   
//                                                                           
//  Copyright: 
//    (C) 2024 Thorsten Brach. All rights reserved                                                                         
//                                                                           
//  Disclaimer:                                                                           
//    This project is provided without any guarantee and can be used for   
//    private and commercial purposes. Any commercial use is at the user’s 
//    own risk and responsibility.
//
// -------------------------------------------------------------------------
VAR_INPUT
  /// Start of the command at the rising edge
  Execute            : BOOL;
  /// Processing Mode
  ProcessingMode     : ProcessingMode;
  /// Specifies the desired byte addresses that shall be read
  Index              : ARRAY[0..4] OF USINT; 
  /// Defines the target sequence in which the command will be executed
  SequenceFlag       : SequenceFlag;
  /// ID of associated trigger function:
  /// •  0: No Trigger (default)  No trigger related behavior
  /// • >0: Trigger - Start executing when the trigger function with the identical EmitterID is triggered.
  /// Always positive.
  /// For more information, see chapter 5.5.12 Triggers
  ListenerID         : SINT;
END_VAR
VAR_OUTPUT
  /// The command has been completed successfully
  Done               : BOOL;
  /// TRUE, while the following outputs return valid values:
  /// • Values
  Valid              : BOOL; 
  /// FB is being processed
  Busy               : BOOL;
  /// Command is transferred and confirmed by the RC
  CommandBuffered    : BOOL;
  /// The command was aborted by another command.
  CommandAborted     : BOOL;
  /// TRUE, while command is interrupted during execution and can be continued
  CommandInterrupted : BOOL;
  /// Receiving of input parameter values has been acknowledged by RC
  ParameterAccepted  : BOOL;
  /// Returned values of digital inputs
  Values             : ARRAY[0..4] OF BYTE;
  /// Unique system-generated ID of the "Action" when the function is triggered.
  /// • >0: The "Action" is started by the trigger function with identical FollowID.
  /// • <0: The "Action" is stopped by the trigger function with identical FollowID.
  /// For more information see chapter 5.5.12.4.
  OriginID           : USINT;
  /// Relates to ListenerID >0 
  /// Number of successful trigger -based command invocations
  /// For more information refer to chapter 5.5.12.4.
  InvocationCounter  : USINT;
END_VAR

                  
                

METHOD PROTECTED OnCall
VAR_IN_OUT
  /// Robot assignment of function
  AxesGroup         : AxesGroup; 
END_VAR
                        
                      
END_METHOD
END_FUNCTION_BLOCK

/// Read digital output group of RC
FUNCTION_BLOCK ReadDigitalOutputsFB EXTENDS RobotLibraryBaseFB
// ------------------------------------------------------------------------- 
//  SRCI Robot Library                                                
// ------------------------------------------------------------------------- 
//                                                                           
//  Object:      ReadDigitalOutputsFB                                       
//  Author:      Thorsten Brach                                                
//  Date:        2024-06-01
//
//  Description:                                              
//   
//                                                                           
//  Copyright: 
//    (C) 2024 Thorsten Brach. All rights reserved                                                                         
//                                                                           
//  Disclaimer:                                                                           
//    This project is provided without any guarantee and can be used for   
//    private and commercial purposes. Any commercial use is at the user’s 
//    own risk and responsibility.
//
// -------------------------------------------------------------------------
VAR_INPUT
  /// Start of the command at the rising edge
  Execute            : BOOL;
  /// Processing Mode
  ProcessingMode     : ProcessingMode;
  /// Specifies the desired byte addresses that shall be read
  Index              : ARRAY[0..4] OF USINT; 
  /// Defines the target sequence in which the command will be executed
  SequenceFlag       : SequenceFlag;
  /// ID of associated trigger function:
  /// •  0: No Trigger (default)  No trigger related behavior
  /// • >0: Trigger - Start executing when the trigger function with the identical EmitterID is triggered.
  /// Always positive.
  /// For more information, see chapter 5.5.12 Triggers
  ListenerID         : SINT;
END_VAR
VAR_OUTPUT
  /// The command has been completed successfully
  Done               : BOOL;
  /// TRUE, while the following outputs return valid values:
  /// • Values
  Valid              : BOOL; 
  /// FB is being processed
  Busy               : BOOL;
  /// Command is transferred and confirmed by the RC
  CommandBuffered    : BOOL;
  /// The command was aborted by another command.
  CommandAborted     : BOOL;
  /// TRUE, while command is interrupted during execution and can be continued
  CommandInterrupted : BOOL;
  /// Receiving of input parameter values has been acknowledged by RC
  ParameterAccepted  : BOOL;
  /// Returned values of digital inputs
  Values             : ARRAY[0..4] OF BYTE;
  /// Unique system-generated ID of the "Action" when the function is triggered.
  /// • >0: The "Action" is started by the trigger function with identical FollowID.
  /// • <0: The "Action" is stopped by the trigger function with identical FollowID.
  /// For more information see chapter 5.5.12.4.
  OriginID           : USINT;
  /// Relates to ListenerID >0 
  /// Number of successful trigger -based command invocations
  /// For more information refer to chapter 5.5.12.4.
  InvocationCounter  : USINT;
END_VAR

                  
                

METHOD PROTECTED OnCall
VAR_IN_OUT
  /// Robot assignment of function
  AxesGroup         : AxesGroup; 
END_VAR
                        
                      
END_METHOD
END_FUNCTION_BLOCK

/// Read content of selected user frame number
FUNCTION_BLOCK ReadFrameDataFB EXTENDS RobotLibraryBaseFB
// ------------------------------------------------------------------------- 
//  SRCI Robot Library                                                
// ------------------------------------------------------------------------- 
//                                                                           
//  Object:      ReadFrameDataFB                                       
//  Author:      Thorsten Brach                                                
//  Date:        2024-06-01
//
//  Description:                                              
//   
//                                                                           
//  Copyright: 
//    (C) 2024 Thorsten Brach. All rights reserved                                                                         
//                                                                           
//  Disclaimer:                                                                           
//    This project is provided without any guarantee and can be used for   
//    private and commercial purposes. Any commercial use is at the user’s 
//    own risk and responsibility.
//
// -------------------------------------------------------------------------
VAR_INPUT
  /// Start of the command at the rising edge
  Execute            : BOOL;
  /// Frame index
  /// • -1: Currently used frame on RC
  /// • 0: WCS
  /// • 1 (default)..254: UCS (User frames)
  FrameNo            : INT;
END_VAR
VAR_OUTPUT
  /// The command has been completed successfully
  Done               : BOOL;
  /// FB is being processed
  Busy               : BOOL;
  /// Command is transferred and confirmed by the RC
  CommandBuffered    : BOOL;
  /// Frame index
  FrameNoReturn      : USINT;
  /// Frame data (see chapter 5.5.6.2)
  FrameData          : FrameData;
END_VAR

                  
                

METHOD PROTECTED OnCall
VAR_IN_OUT
  /// Robot assignment of function
  AxesGroup         : AxesGroup; 
END_VAR
                        
                      
END_METHOD
END_FUNCTION_BLOCK

